TYPE ST_HVFASystemDefaultParameters :
STRUCT
	aSetPointLimitsTemperature : ARRAY[1..2] OF REAL := [10,28];
END_STRUCT
END_TYPE

(* stored: Version 1.1.0.1, ProductVersion 3.1.4024.9
   DUT ST_HVFASystemDefaultParameters: Id {19ecbe41-1a31-47dc-a36b-1ab9ec637190} *)
